// TwinCAT 3 PLC project rixs_optics
// ProgramVersion: 3.1.4022.7
// libraries:
//   lcls2-cc-lib, * (SLAC)
//   PMPS, * (SLAC - LCLS)
//   Tc2_MC2, * (Beckhoff Automation GmbH)
//   Tc2_SerialCom, * (Beckhoff Automation GmbH)
//   Tc2_Standard, * (Beckhoff Automation GmbH)
//   Tc2_System, * (Beckhoff Automation GmbH)
//   Tc2_Utilities, * (Beckhoff Automation GmbH)
//   Tc3_Module, * (Beckhoff Automation GmbH)
//   LCLS General,newest,SLAC
//   lcls-twincat-motion,newest,SLAC
//   lcls-twincat-optics,newest,SLAC
// project tree:
//   DUTs/ ENUM_XS_YAG_States.TcDUT (not stored)
//   Function Blocks/ FB_XS_YAG_States.TcPOU (not stored)
//   GVLs/ GVL_COM_Buffers.TcGVL (not stored), GVL_M1K1.TcGVL (not stored), GVL_M1K1_BENDER_Constants.TcGVL (not stored), GVL_M1K1_BENDER_RTD.TcGVL (not stored), GVL_M1K1_Constants.TcGVL (not stored), GVL_M1K2.TcGVL (not stored), GVL_M1K2_Constants.TcGVL (not stored), GVL_PMPS.TcGVL (not stored), GVL_SerialIO.TcGVL (not stored), Main.TcGVL
//   / PiezoDriver.TcTTO (not stored), PlcTask.TcTTO (not stored), SerialIO.TcTTO (not stored)
//   POUs/ PRG_1_PlcTask.TcPOU (not stored), PRG_2_PMPS_POST.TcPOU (not stored), PRG_MR1K1_BEND.TcPOU (not stored), PRG_MR1K1_BEND_BENDER.TcPOU (not stored), PRG_MR1K2_SWITCH.TcPOU (not stored), PRG_SL1K2_EXIT.TcPOU (not stored), PRG_SP1K1_MONO.TcPOU (not stored), PRG_SPO_PMPS.TcPOU, PRG_ST1K1_ZOS.TcPOU (not stored)
//   POUs/Serial Comm/ PiezoSerial.TcPOU (not stored), P_Serial_Com.TcPOU (not stored)
// real-time tasks:
//   TASK PlcTask: cycle T#10ms, priority 20, ADS port 350
//   TASK PiezoDriver: cycle T#1ms, priority 3, ADS port 351
//   TASK SerialIO: cycle T#2ms, priority 1, ADS port 352
// motion (NC):
// I/O:
//   DEVICE Device 1 (EtherCAT)
// variable links:
//   rixs_optics Instance <-> Device 1 (EtherCAT)/Term 1 (EK1200)/E5 (EK1122)/Box 84 (EP2338-0002)
//     PlcTask Outputs/PRG_SP1K1_MONO.bLEDPower01 <-> Channel 10/Output
//     PlcTask Outputs/PRG_SP1K1_MONO.bLEDPower02 <-> Channel 12/Output
//     PlcTask Outputs/PRG_SP1K1_MONO.bLEDPower03 <-> Channel 14/Output
//   rixs_optics Instance <-> Device 1 (EtherCAT)/Term 1 (EK1200)/E5 (EK1122)/SL1K2-EXIT (EK1100)/EL2004_SL1K2
//     PlcTask Outputs/PRG_SL1K2_EXIT.bFanOn <-> Channel 1/Output
//     PlcTask Outputs/PRG_SL1K2_EXIT.bLEDPower <-> Channel 2/Output
//     PlcTask Outputs/PRG_SL1K2_EXIT.fbGige.bGigePower <-> Channel 3/Output
//   rixs_optics Instance <-> Device 1 (EtherCAT)/Term 1 (EK1200)/E5 (EK1122)/SL1K2-EXIT (EK1100)/EL3201_SL1K2_1
//     PlcTask Inputs/PRG_SL1K2_EXIT.RTD_Crystal_TOP.bOverrange <-> RTD/Status/Overrange
//     PlcTask Inputs/PRG_SL1K2_EXIT.RTD_Crystal_TOP.bUnderrange <-> RTD/Status/Underrange
//     PlcTask Inputs/PRG_SL1K2_EXIT.RTD_Crystal_TOP.iRaw <-> RTD/Value
//   rixs_optics Instance <-> Device 1 (EtherCAT)/Term 1 (EK1200)/E5 (EK1122)/SL1K2-EXIT (EK1100)/EL3201_SL1K2_2
//     PlcTask Inputs/PRG_SL1K2_EXIT.RTD_Crystal_BOTTOM.bOverrange <-> RTD/Status/Overrange
//     PlcTask Inputs/PRG_SL1K2_EXIT.RTD_Crystal_BOTTOM.bUnderrange <-> RTD/Status/Underrange
//     PlcTask Inputs/PRG_SL1K2_EXIT.RTD_Crystal_BOTTOM.iRaw <-> RTD/Value
//   rixs_optics Instance <-> Device 1 (EtherCAT)/Term 1 (EK1200)/E5 (EK1122)/SL1K2-EXIT (EK1100)/EL3201_SL1K2_3
//     PlcTask Inputs/PRG_SL1K2_EXIT.RTD_YAG.bOverrange <-> RTD/Status/Overrange
//     PlcTask Inputs/PRG_SL1K2_EXIT.RTD_YAG.bUnderrange <-> RTD/Status/Underrange
//     PlcTask Inputs/PRG_SL1K2_EXIT.RTD_YAG.iRaw <-> RTD/Value
//   rixs_optics Instance <-> Device 1 (EtherCAT)/Term 1 (EK1200)/E5 (EK1122)/SL1K2-EXIT (EK1100)/EL3201_SL1K2_4
//     PlcTask Inputs/PRG_SL1K2_EXIT.RTD_HeatSync.bOverrange <-> RTD/Status/Overrange
//     PlcTask Inputs/PRG_SL1K2_EXIT.RTD_HeatSync.bUnderrange <-> RTD/Status/Underrange
//     PlcTask Inputs/PRG_SL1K2_EXIT.RTD_HeatSync.iRaw <-> RTD/Value
//   rixs_optics Instance <-> Device 1 (EtherCAT)/Term 1 (EK1200)/E5 (EK1122)/SL1K2-EXIT (EK1100)/EL4004_SL1K2
//     PlcTask Outputs/PRG_SL1K2_EXIT.fbGige.iIlluminatorINT <-> AO Outputs Channel 1/Analog output
//   rixs_optics Instance <-> Device 1 (EtherCAT)/Term 1 (EK1200)/E5 (EK1122)/SL1K2-EXIT (EK1100)/EL5042_SL1K2_PITCH_VERT
//     PlcTask Inputs/Main.M19.nRawEncoderUINT <-> FB Inputs Channel 1/Position
//     PlcTask Inputs/Main.M20.nRawEncoderUINT <-> FB Inputs Channel 2/Position
//   rixs_optics Instance <-> Device 1 (EtherCAT)/Term 1 (EK1200)/E5 (EK1122)/SL1K2-EXIT (EK1100)/EL5042_SL1K2_ROLL_GAP
//     PlcTask Inputs/Main.M21.nRawEncoderUINT <-> FB Inputs Channel 1/Position
//     PlcTask Inputs/Main.M22.nRawEncoderUINT <-> FB Inputs Channel 2/Position
//   rixs_optics Instance <-> Device 1 (EtherCAT)/Term 1 (EK1200)/E5 (EK1122)/SL1K2-EXIT (EK1100)/EL5042_SL1K2_YAG
//     PlcTask Inputs/Main.M23.nRawEncoderUINT <-> FB Inputs Channel 1/Position
//   rixs_optics Instance <-> Device 1 (EtherCAT)/Term 1 (EK1200)/E5 (EK1122)/SL1K2-EXIT (EK1100)/EL7047_SL1K2_GAP
//     PlcTask Inputs/Main.M22.bLimitBackwardEnable <-> STM Status/Status/Digital input 1
//     PlcTask Inputs/Main.M22.bLimitForwardEnable <-> STM Status/Status/Digital input 2
//   rixs_optics Instance <-> Device 1 (EtherCAT)/Term 1 (EK1200)/E5 (EK1122)/SL1K2-EXIT (EK1100)/EL7047_SL1K2_PITCH
//     PlcTask Inputs/Main.M19.bLimitBackwardEnable <-> STM Status/Status/Digital input 1
//     PlcTask Inputs/Main.M19.bLimitForwardEnable <-> STM Status/Status/Digital input 2
//   rixs_optics Instance <-> Device 1 (EtherCAT)/Term 1 (EK1200)/E5 (EK1122)/SL1K2-EXIT (EK1100)/EL7047_SL1K2_ROLL
//     PlcTask Inputs/Main.M21.bLimitBackwardEnable <-> STM Status/Status/Digital input 1
//     PlcTask Inputs/Main.M21.bLimitForwardEnable <-> STM Status/Status/Digital input 2
//   rixs_optics Instance <-> Device 1 (EtherCAT)/Term 1 (EK1200)/E5 (EK1122)/SL1K2-EXIT (EK1100)/EL7047_SL1K2_VERT
//     PlcTask Inputs/Main.M20.bLimitBackwardEnable <-> STM Status/Status/Digital input 2
//     PlcTask Inputs/Main.M20.bLimitForwardEnable <-> STM Status/Status/Digital input 1
//   rixs_optics Instance <-> Device 1 (EtherCAT)/Term 1 (EK1200)/E5 (EK1122)/SL1K2-EXIT (EK1100)/EL7047_SL1K2_YAG
//     PlcTask Inputs/Main.M23.bLimitBackwardEnable <-> STM Status/Status/Digital input 2
//     PlcTask Inputs/Main.M23.bLimitForwardEnable <-> STM Status/Status/Digital input 1
//   rixs_optics Instance <-> Device 1 (EtherCAT)/Term 1 (EK1200)/E5 (EK1122)/X1 SP1K1-MONO(EK1100)/SP1K1-EL1004-E17
//     PlcTask Inputs/PRG_SP1K1_MONO.bSTOEnable1 <-> Channel 1/Input
//     PlcTask Inputs/PRG_SP1K1_MONO.bSTOEnable2 <-> Channel 2/Input
//   rixs_optics Instance <-> Device 1 (EtherCAT)/Term 1 (EK1200)/E5 (EK1122)/X1 SP1K1-MONO(EK1100)/SP1K1-EL3054-E12
//     PlcTask Inputs/PRG_SP1K1_MONO.flow_1 <-> AI Standard Channel 1/Value
//     PlcTask Inputs/PRG_SP1K1_MONO.flow_2 <-> AI Standard Channel 2/Value
//     PlcTask Inputs/PRG_SP1K1_MONO.pres_1 <-> AI Standard Channel 3/Value
//   rixs_optics Instance <-> Device 1 (EtherCAT)/Term 1 (EK1200)/E5 (EK1122)/X1 SP1K1-MONO(EK1100)/SP1K1-EL3202-E13
//     PlcTask Inputs/PRG_SP1K1_MONO.RTD1.bError <-> RTD Inputs Channel 1/Status/Error
//     PlcTask Inputs/PRG_SP1K1_MONO.RTD2.bError <-> RTD Inputs Channel 2/Status/Error
//     PlcTask Inputs/PRG_SP1K1_MONO.RTD1.bOverrange <-> RTD Inputs Channel 1/Status/Overrange
//     PlcTask Inputs/PRG_SP1K1_MONO.RTD2.bOverrange <-> RTD Inputs Channel 2/Status/Overrange
//     PlcTask Inputs/PRG_SP1K1_MONO.RTD1.bUnderrange <-> RTD Inputs Channel 1/Status/Underrange
//     PlcTask Inputs/PRG_SP1K1_MONO.RTD2.bUnderrange <-> RTD Inputs Channel 2/Status/Underrange
//     PlcTask Inputs/PRG_SP1K1_MONO.RTD1.iRaw <-> RTD Inputs Channel 1/Value
//     PlcTask Inputs/PRG_SP1K1_MONO.RTD2.iRaw <-> RTD Inputs Channel 2/Value
//   rixs_optics Instance <-> Device 1 (EtherCAT)/Term 1 (EK1200)/E5 (EK1122)/X1 SP1K1-MONO(EK1100)/SP1K1-EL3202-E14
//     PlcTask Inputs/PRG_SP1K1_MONO.RTD3.bError <-> RTD Inputs Channel 1/Status/Error
//     PlcTask Inputs/PRG_SP1K1_MONO.RTD4.bError <-> RTD Inputs Channel 2/Status/Error
//     PlcTask Inputs/PRG_SP1K1_MONO.RTD3.bOverrange <-> RTD Inputs Channel 1/Status/Overrange
//     PlcTask Inputs/PRG_SP1K1_MONO.RTD4.bOverrange <-> RTD Inputs Channel 2/Status/Overrange
//     PlcTask Inputs/PRG_SP1K1_MONO.RTD3.bUnderrange <-> RTD Inputs Channel 1/Status/Underrange
//     PlcTask Inputs/PRG_SP1K1_MONO.RTD4.bUnderrange <-> RTD Inputs Channel 2/Status/Underrange
//     PlcTask Inputs/PRG_SP1K1_MONO.RTD3.iRaw <-> RTD Inputs Channel 1/Value
//     PlcTask Inputs/PRG_SP1K1_MONO.RTD4.iRaw <-> RTD Inputs Channel 2/Value
//   rixs_optics Instance <-> Device 1 (EtherCAT)/Term 1 (EK1200)/E5 (EK1122)/X1 SP1K1-MONO(EK1100)/SP1K1-EL3204-E15
//     PlcTask Inputs/PRG_SP1K1_MONO.RTD5.bError <-> RTD Inputs Channel 1/Status/Error
//     PlcTask Inputs/PRG_SP1K1_MONO.RTD6.bError <-> RTD Inputs Channel 2/Status/Error
//     PlcTask Inputs/PRG_SP1K1_MONO.RTD5.bOverrange <-> RTD Inputs Channel 1/Status/Overrange
//     PlcTask Inputs/PRG_SP1K1_MONO.RTD6.bOverrange <-> RTD Inputs Channel 2/Status/Overrange
//     PlcTask Inputs/PRG_SP1K1_MONO.RTD5.bUnderrange <-> RTD Inputs Channel 1/Status/Underrange
//     PlcTask Inputs/PRG_SP1K1_MONO.RTD6.bUnderrange <-> RTD Inputs Channel 2/Status/Underrange
//     PlcTask Inputs/PRG_SP1K1_MONO.RTD5.iRaw <-> RTD Inputs Channel 1/Value
//     PlcTask Inputs/PRG_SP1K1_MONO.RTD6.iRaw <-> RTD Inputs Channel 2/Value
//   rixs_optics Instance <-> Device 1 (EtherCAT)/Term 1 (EK1200)/E5 (EK1122)/X1 SP1K1-MONO(EK1100)/SP1K1-EL3204-E16
//     PlcTask Inputs/PRG_SP1K1_MONO.RTD7.bError <-> RTD Inputs Channel 1/Status/Error
//     PlcTask Inputs/PRG_SP1K1_MONO.RTD8.bError <-> RTD Inputs Channel 2/Status/Error
//     PlcTask Inputs/PRG_SP1K1_MONO.RTD7.bOverrange <-> RTD Inputs Channel 1/Status/Overrange
//     PlcTask Inputs/PRG_SP1K1_MONO.RTD8.bOverrange <-> RTD Inputs Channel 2/Status/Overrange
//     PlcTask Inputs/PRG_SP1K1_MONO.RTD7.bUnderrange <-> RTD Inputs Channel 1/Status/Underrange
//     PlcTask Inputs/PRG_SP1K1_MONO.RTD8.bUnderrange <-> RTD Inputs Channel 2/Status/Underrange
//     PlcTask Inputs/PRG_SP1K1_MONO.RTD7.iRaw <-> RTD Inputs Channel 1/Value
//     PlcTask Inputs/PRG_SP1K1_MONO.RTD8.iRaw <-> RTD Inputs Channel 2/Value
//   rixs_optics Instance <-> Device 1 (EtherCAT)/Term 1 (EK1200)/E5 (EK1122)/X1 SP1K1-MONO(EK1100)/g_h_m
//     PlcTask Inputs/Main.M9.bLimitBackwardEnable <-> STM Status/Status/Digital input 2
//     PlcTask Inputs/Main.M9.bLimitForwardEnable <-> STM Status/Status/Digital input 1
//   rixs_optics Instance <-> Device 1 (EtherCAT)/Term 1 (EK1200)/E5 (EK1122)/X1 SP1K1-MONO(EK1100)/g_pi_m
//     PlcTask Inputs/Main.M7.bLimitBackwardEnable <-> STM Status/Status/Digital input 2
//     PlcTask Inputs/Main.M7.bLimitForwardEnable <-> STM Status/Status/Digital input 1
//   rixs_optics Instance <-> Device 1 (EtherCAT)/Term 1 (EK1200)/E5 (EK1122)/X1 SP1K1-MONO(EK1100)/g_pi_up_dwn_e
//     PlcTask Inputs/PRG_SP1K1_MONO.gpi_upe/Count <-> FB Inputs Channel 1/Position
//   rixs_optics Instance <-> Device 1 (EtherCAT)/Term 1 (EK1200)/E5 (EK1122)/X1 SP1K1-MONO(EK1100)/m_h_m
//     PlcTask Inputs/Main.M8.bLimitBackwardEnable <-> STM Status/Status/Digital input 2
//     PlcTask Inputs/Main.M8.bLimitForwardEnable <-> STM Status/Status/Digital input 1
//   rixs_optics Instance <-> Device 1 (EtherCAT)/Term 1 (EK1200)/E5 (EK1122)/X1 SP1K1-MONO(EK1100)/m_pi_m
//     PlcTask Inputs/Main.M6.bLimitBackwardEnable <-> STM Status/Status/Digital input 2
//     PlcTask Inputs/Main.M6.bLimitForwardEnable <-> STM Status/Status/Digital input 1
//   rixs_optics Instance <-> Device 1 (EtherCAT)/Term 1 (EK1200)/E5 (EK1122)/X1 SP1K1-MONO(EK1100)/m_pi_up_dwn_e
//     PlcTask Inputs/PRG_SP1K1_MONO.mpi_upe/Count <-> FB Inputs Channel 1/Position
//   rixs_optics Instance <-> Device 1 (EtherCAT)/Term 1 (EK1200)/E5 (EK1122)/X1 SP1K1-MONO(EK1100)/s_io_m
//     PlcTask Inputs/Main.M10.bLimitBackwardEnable <-> STM Status/Status/Digital input 2
//     PlcTask Inputs/Main.M10.bLimitForwardEnable <-> STM Status/Status/Digital input 1
//     PlcTask Inputs/Main.sio_current <-> STM Synchron info data/Info data 1
//     PlcTask Inputs/Main.sio_load <-> STM Synchron info data/Info data 2
//   rixs_optics Instance <-> Device 1 (EtherCAT)/Term 1 (EK1200)/PMPS_FFO
//     PlcTask Outputs/GVL_PMPS.fbFastFaultOutput1.q_xFastFaultOut <-> Channel 1/Output
//     PlcTask Outputs/GVL_PMPS.fbFastFaultOutput2.q_xFastFaultOut <-> Channel 2/Output
//   rixs_optics Instance <-> Device 1 (EtherCAT)/Term 1 (EK1200)/PMPS_PRE
//     PlcTask Inputs/PRG_2_PMPS_POST.fbArbiterIO.i_stCurrentBP <-> IO Inputs/CurrentBP
//     PlcTask Inputs/PRG_2_PMPS_POST.fbArbiterIO.xTxPDO_state <-> SYNC Inputs/TxPDO state
//     PlcTask Inputs/PRG_2_PMPS_POST.fbArbiterIO.xTxPDO_toggle <-> SYNC Inputs/TxPDO toggle
//     PlcTask Outputs/PRG_2_PMPS_POST.fbArbiterIO.q_stRequestedBP <-> IO Outputs/RequestedBP
//     PlcTask Outputs/PRG_MR1K1_BEND.nMR1K1_Y_ENC_PMPS <-> IO Outputs/MR1K1_Y_ENC
//   rixs_optics Instance <-> Device 1 (EtherCAT)/Term 1 (EK1200)/Term 5 (EK1122)/EK1100_M1K2/EL1004_M1K2_STO
//     PlcTask Inputs/PRG_MR1K2_SWITCH.M1K2.fbRunHOMS.bSTOEnable1 <-> Channel 1/Input
//     PlcTask Inputs/PRG_MR1K2_SWITCH.M1K2.fbRunHOMS.bSTOEnable2 <-> Channel 2/Input
//   rixs_optics Instance <-> Device 1 (EtherCAT)/Term 1 (EK1200)/Term 5 (EK1122)/EK1100_M1K2/EL5042_M1K2_Pitch
//     PlcTask Inputs/GVL_M1K1.M1K1_Pitch.diEncCnt <-> FB Inputs Channel 1/Position
//     PlcTask Inputs/GVL_M1K2.M1K2_Pitch.diEncCnt <-> FB Inputs Channel 1/Position
//   rixs_optics Instance <-> Device 1 (EtherCAT)/Term 1 (EK1200)/Term 5 (EK1122)/EK1100_M1K2/EL5042_M1K2_Xupdwn
//     PlcTask Inputs/PRG_MR1K2_SWITCH.M1K2.fbRunHOMS.stXdwnEnc/Count <-> FB Inputs Channel 2/Position
//     PlcTask Inputs/PRG_MR1K2_SWITCH.M1K2.fbRunHOMS.stXupEnc/Count <-> FB Inputs Channel 1/Position
//   rixs_optics Instance <-> Device 1 (EtherCAT)/Term 1 (EK1200)/Term 5 (EK1122)/EK1100_M1K2/EL5042_M1K2_Yleftright
//     PlcTask Inputs/PRG_MR1K2_SWITCH.M1K2.fbRunHOMS.stYdwnEnc/Count <-> FB Inputs Channel 2/Position
//     PlcTask Inputs/PRG_MR1K2_SWITCH.M1K2.fbRunHOMS.stYupEnc/Count <-> FB Inputs Channel 1/Position
//   rixs_optics Instance <-> Device 1 (EtherCAT)/Term 1 (EK1200)/Term 5 (EK1122)/EK1100_M1K2/EL6001_M1K2_PitchFine
//     SerialIO Inputs/GVL_SerialIO.Serial_stComIn_M1K2/D[{0..21}] <-> COM Inputs/Data In {0..21}  (22 links)
//     SerialIO Inputs/GVL_SerialIO.Serial_stComIn_M1K2/Status <-> COM Inputs/Status
//     SerialIO Outputs/GVL_SerialIO.Serial_stComOut_M1K2/Ctrl <-> COM Outputs/Ctrl
//     SerialIO Outputs/GVL_SerialIO.Serial_stComOut_M1K2/D[{0..21}] <-> COM Outputs/Data Out {0..21}  (22 links)
//   rixs_optics Instance <-> Device 1 (EtherCAT)/Term 1 (EK1200)/Term 5 (EK1122)/EK1100_M1K2/EL7047_M1K2_PitchCoarse
//     PlcTask Inputs/Main.M5.bLimitBackwardEnable <-> STM Status/Status/Digital input 2
//     PlcTask Inputs/Main.M5.bLimitForwardEnable <-> STM Status/Status/Digital input 1
//   rixs_optics Instance <-> Device 1 (EtherCAT)/Term 1 (EK1200)/Term 5 (EK1122)/EK1100_M1K2/EL7047_M1K2_Xdwn
//     PlcTask Inputs/Main.M4.bLimitBackwardEnable <-> STM Status/Status/Digital input 2
//     PlcTask Inputs/Main.M4.bLimitForwardEnable <-> STM Status/Status/Digital input 1
//   rixs_optics Instance <-> Device 1 (EtherCAT)/Term 1 (EK1200)/Term 5 (EK1122)/EK1100_M1K2/EL7047_M1K2_Xup
//     PlcTask Inputs/Main.M3.bLimitBackwardEnable <-> STM Status/Status/Digital input 2
//     PlcTask Inputs/Main.M3.bLimitForwardEnable <-> STM Status/Status/Digital input 1
//   rixs_optics Instance <-> Device 1 (EtherCAT)/Term 1 (EK1200)/Term 5 (EK1122)/EK1100_M1K2/EL7047_M1K2_Yleft
//     PlcTask Inputs/Main.M1.bLimitBackwardEnable <-> STM Status/Status/Digital input 2
//     PlcTask Inputs/Main.M1.bLimitForwardEnable <-> STM Status/Status/Digital input 1
//   rixs_optics Instance <-> Device 1 (EtherCAT)/Term 1 (EK1200)/Term 5 (EK1122)/EK1100_M1K2/EL7047_M1K2_Yright
//     PlcTask Inputs/Main.M2.bLimitBackwardEnable <-> STM Status/Status/Digital input 2
//     PlcTask Inputs/Main.M2.bLimitForwardEnable <-> STM Status/Status/Digital input 1
//   rixs_optics Instance <-> Device 1 (EtherCAT)/Term 1 (EK1200)/Term 5 (EK1122)/EK1100_MR1K1/EL1004_M1K1_STO
//     PlcTask Inputs/PRG_MR1K1_BEND.M1K1.fbRunHOMS.bSTOEnable1 <-> Channel 1/Input
//     PlcTask Inputs/PRG_MR1K1_BEND.M1K1.fbRunHOMS.bSTOEnable2 <-> Channel 2/Input
//   rixs_optics Instance <-> Device 1 (EtherCAT)/Term 1 (EK1200)/Term 5 (EK1122)/EK1100_MR1K1/EL5042_M1K1_Xupdwn
//     PlcTask Inputs/PRG_MR1K1_BEND.M1K1.fbRunHOMS.stXdwnEnc/Count <-> FB Inputs Channel 2/Position
//     PlcTask Inputs/PRG_MR1K1_BEND.M1K1.fbRunHOMS.stXupEnc/Count <-> FB Inputs Channel 1/Position
//   rixs_optics Instance <-> Device 1 (EtherCAT)/Term 1 (EK1200)/Term 5 (EK1122)/EK1100_MR1K1/EL5042_M1K1_Yupdwn
//     PlcTask Inputs/PRG_MR1K1_BEND.M1K1.fbRunHOMS.stYdwnEnc/Count <-> FB Inputs Channel 2/Position
//     PlcTask Inputs/PRG_MR1K1_BEND.M1K1.fbRunHOMS.stYupEnc/Count <-> FB Inputs Channel 1/Position
//     PlcTask Inputs/PRG_MR1K1_BEND.bMR1K1_Y_ENC_Ready <-> FB Inputs Channel 1/Status/Ready
//     PlcTask Inputs/PRG_MR1K1_BEND.bMR1K1_Y_ENC_TxPDO <-> FB Inputs Channel 1/Status/TxPDO State
//   rixs_optics Instance <-> Device 1 (EtherCAT)/Term 1 (EK1200)/Term 5 (EK1122)/EK1100_MR1K1/EL7047_M1K1_PitchCoarse
//     PlcTask Inputs/Main.M16.bLimitBackwardEnable <-> STM Status/Status/Digital input 2
//     PlcTask Inputs/Main.M16.bLimitForwardEnable <-> STM Status/Status/Digital input 1
//   rixs_optics Instance <-> Device 1 (EtherCAT)/Term 1 (EK1200)/Term 5 (EK1122)/EK1100_MR1K1/EL7047_M1K1_Xdwn
//     PlcTask Inputs/Main.M15.bLimitBackwardEnable <-> STM Status/Status/Digital input 2
//     PlcTask Inputs/Main.M15.bLimitForwardEnable <-> STM Status/Status/Digital input 1
//   rixs_optics Instance <-> Device 1 (EtherCAT)/Term 1 (EK1200)/Term 5 (EK1122)/EK1100_MR1K1/EL7047_M1K1_Xup
//     PlcTask Inputs/Main.M14.bLimitBackwardEnable <-> STM Status/Status/Digital input 2
//     PlcTask Inputs/Main.M14.bLimitForwardEnable <-> STM Status/Status/Digital input 1
//   rixs_optics Instance <-> Device 1 (EtherCAT)/Term 1 (EK1200)/Term 5 (EK1122)/EK1100_MR1K1/EL7047_M1K1_Ydwn
//     PlcTask Inputs/Main.M12.bLimitBackwardEnable <-> STM Status/Status/Digital input 2
//     PlcTask Inputs/Main.M13.bLimitBackwardEnable <-> STM Status/Status/Digital input 2
//     PlcTask Inputs/Main.M13.bLimitForwardEnable <-> STM Status/Status/Digital input 1
//   rixs_optics Instance <-> Device 1 (EtherCAT)/Term 1 (EK1200)/Term 5 (EK1122)/EK1100_MR1K1/EL7047_M1K1_Yup
//     PlcTask Inputs/Main.M12.bLimitForwardEnable <-> STM Status/Status/Digital input 1
//   rixs_optics Instance <-> Device 1 (EtherCAT)/Term 1 (EK1200)/Term 5 (EK1122)/EK1100_MR1K1_BEND/EL1004_M1K1_BENDER_STO
//     PlcTask Inputs/PRG_MR1K1_BEND_BENDER.M1K1BENDbSTOEnable1 <-> Channel 1/Input
//     PlcTask Inputs/PRG_MR1K1_BEND_BENDER.M1K1BENDbSTOEnable2 <-> Channel 2/Input
//   rixs_optics Instance <-> Device 1 (EtherCAT)/Term 1 (EK1200)/Term 5 (EK1122)/EK1100_MR1K1_BEND/EL2024-0010_M1K1_BEND_LED1
//     PlcTask Outputs/PRG_MR1K1_BEND.bLEDPower01 <-> Channel 1/Output
//     PlcTask Outputs/PRG_MR1K1_BEND.bLEDPower02 <-> Channel 2/Output
//     PlcTask Outputs/PRG_MR1K1_BEND.bLEDPower03 <-> Channel 3/Output
//     PlcTask Outputs/PRG_MR1K1_BEND.bLEDPower04 <-> Channel 4/Output
//   rixs_optics Instance <-> Device 1 (EtherCAT)/Term 1 (EK1200)/Term 5 (EK1122)/EK1100_MR1K1_BEND/EL3202-0010_M1K1DS2_M1K1DS3
//     PlcTask Inputs/GVL_M1K1_BENDER_RTD.nM1K1DS_RTD_2 <-> RTD Inputs Channel 1/Value
//     PlcTask Inputs/GVL_M1K1_BENDER_RTD.nM1K1DS_RTD_3 <-> RTD Inputs Channel 2/Value
//   rixs_optics Instance <-> Device 1 (EtherCAT)/Term 1 (EK1200)/Term 5 (EK1122)/EK1100_MR1K1_BEND/EL3202-0010_M1K1US1_M1K1US2
//     PlcTask Inputs/GVL_M1K1_BENDER_RTD.nM1K1US_RTD_1 <-> RTD Inputs Channel 1/Value
//     PlcTask Inputs/GVL_M1K1_BENDER_RTD.nM1K1US_RTD_2 <-> RTD Inputs Channel 2/Value
//   rixs_optics Instance <-> Device 1 (EtherCAT)/Term 1 (EK1200)/Term 5 (EK1122)/EK1100_MR1K1_BEND/EL3202-0010_M1K1US3_M1K1DS1
//     PlcTask Inputs/GVL_M1K1_BENDER_RTD.nM1K1DS_RTD_1 <-> RTD Inputs Channel 2/Value
//     PlcTask Inputs/GVL_M1K1_BENDER_RTD.nM1K1US_RTD_3 <-> RTD Inputs Channel 1/Value
//   rixs_optics Instance <-> Device 1 (EtherCAT)/Term 1 (EK1200)/Term 5 (EK1122)/EK1100_MR1K1_BEND/EL5042_M1K1_BEND_USDS
//     PlcTask Inputs/Main.M17.nRawEncoderULINT <-> FB Inputs Channel 1/Position
//     PlcTask Inputs/Main.M18.nRawEncoderULINT <-> FB Inputs Channel 2/Position
//   rixs_optics Instance <-> Device 1 (EtherCAT)/Term 1 (EK1200)/Term 5 (EK1122)/EK1100_MR1K1_BEND/EL7041_M1K1_BEND_DS
//     PlcTask Inputs/Main.M18.bLimitBackwardEnable <-> STM Status/Status/Digital input 2
//     PlcTask Inputs/Main.M18.bLimitForwardEnable <-> STM Status/Status/Digital input 1
//   rixs_optics Instance <-> Device 1 (EtherCAT)/Term 1 (EK1200)/Term 5 (EK1122)/EK1100_MR1K1_BEND/EL7041_M1K1_BEND_US
//     PlcTask Inputs/Main.M17.bLimitBackwardEnable <-> STM Status/Status/Digital input 2
//     PlcTask Inputs/Main.M17.bLimitForwardEnable <-> STM Status/Status/Digital input 1
//   rixs_optics Instance <-> Device 1 (EtherCAT)/Term 1 (EK1200)/Term 5 (EK1122)/EK1100_ST1K2_ZOS/ST1K1-EL2008
//     PlcTask Outputs/Main.M24.bBrakeRelease <-> Channel 1/Output
//   rixs_optics Instance <-> Device 1 (EtherCAT)/Term 1 (EK1200)/Term 5 (EK1122)/EK1100_ST1K2_ZOS/ST1K1-EL7041
//     PlcTask Inputs/Main.M24.bLimitBackwardEnable <-> STM Status/Status/Digital input 2
//     PlcTask Inputs/Main.M24.bLimitForwardEnable <-> STM Status/Status/Digital input 1
//   rixs_optics Instance <-> NC-Task 1 SAF/Axes/Axis 24 ST1K1-ZOS-MMS
//     PlcTask Inputs/Main.M24.Axis.NcToPlc <-> Outputs/ToPlc
//     PlcTask Outputs/Main.M24.Axis.PlcToNc <-> Inputs/FromPlc
//   rixs_optics Instance <-> NC-Task 1 SAF/Axes/M1K1-BEND-DS
//     PlcTask Inputs/Main.M18.Axis.NcToPlc <-> Outputs/ToPlc
//     PlcTask Outputs/Main.M18.Axis.PlcToNc <-> Inputs/FromPlc
//   rixs_optics Instance <-> NC-Task 1 SAF/Axes/M1K1-BEND-US
//     PlcTask Inputs/Main.M17.Axis.NcToPlc <-> Outputs/ToPlc
//     PlcTask Outputs/Main.M17.Axis.PlcToNc <-> Inputs/FromPlc
//   rixs_optics Instance <-> NC-Task 1 SAF/Axes/M1K1-Pitch
//     PlcTask Inputs/Main.M16.Axis.NcToPlc <-> Outputs/ToPlc
//     PlcTask Outputs/Main.M16.Axis.PlcToNc <-> Inputs/FromPlc
//   rixs_optics Instance <-> NC-Task 1 SAF/Axes/M1K1-Xdwn
//     PlcTask Inputs/Main.M15.Axis.NcToPlc <-> Outputs/ToPlc
//     PlcTask Outputs/Main.M15.Axis.PlcToNc <-> Inputs/FromPlc
//   rixs_optics Instance <-> NC-Task 1 SAF/Axes/M1K1-Xup
//     PlcTask Inputs/Main.M14.Axis.NcToPlc <-> Outputs/ToPlc
//     PlcTask Outputs/Main.M14.Axis.PlcToNc <-> Inputs/FromPlc
//   rixs_optics Instance <-> NC-Task 1 SAF/Axes/M1K1-Ydwn
//     PlcTask Inputs/Main.M13.Axis.NcToPlc <-> Outputs/ToPlc
//     PlcTask Outputs/Main.M13.Axis.PlcToNc <-> Inputs/FromPlc
//   rixs_optics Instance <-> NC-Task 1 SAF/Axes/M1K1-Yup
//     PlcTask Inputs/Main.M12.Axis.NcToPlc <-> Outputs/ToPlc
//     PlcTask Outputs/Main.M12.Axis.PlcToNc <-> Inputs/FromPlc
//   rixs_optics Instance <-> NC-Task 1 SAF/Axes/M1K2-Pitch
//     PlcTask Inputs/Main.M5.Axis.NcToPlc <-> Outputs/ToPlc
//     PlcTask Outputs/Main.M5.Axis.PlcToNc <-> Inputs/FromPlc
//   rixs_optics Instance <-> NC-Task 1 SAF/Axes/M1K2-Xdwn
//     PlcTask Inputs/Main.M4.Axis.NcToPlc <-> Outputs/ToPlc
//     PlcTask Outputs/Main.M4.Axis.PlcToNc <-> Inputs/FromPlc
//   rixs_optics Instance <-> NC-Task 1 SAF/Axes/M1K2-Xup
//     PlcTask Inputs/Main.M3.Axis.NcToPlc <-> Outputs/ToPlc
//     PlcTask Outputs/Main.M3.Axis.PlcToNc <-> Inputs/FromPlc
//   rixs_optics Instance <-> NC-Task 1 SAF/Axes/M1K2-Yleft
//     PlcTask Inputs/Main.M1.Axis.NcToPlc <-> Outputs/ToPlc
//     PlcTask Outputs/Main.M1.Axis.PlcToNc <-> Inputs/FromPlc
//   rixs_optics Instance <-> NC-Task 1 SAF/Axes/M1K2-Yright
//     PlcTask Inputs/Main.M2.Axis.NcToPlc <-> Outputs/ToPlc
//     PlcTask Outputs/Main.M2.Axis.PlcToNc <-> Inputs/FromPlc
//   rixs_optics Instance <-> NC-Task 1 SAF/Axes/SL1K2-CrystalGap-M22
//     PlcTask Inputs/Main.M22.Axis.NcToPlc <-> Outputs/ToPlc
//     PlcTask Outputs/Main.M22.Axis.PlcToNc <-> Inputs/FromPlc
//   rixs_optics Instance <-> NC-Task 1 SAF/Axes/SL1K2-Pitch-M19
//     PlcTask Inputs/Main.M19.Axis.NcToPlc <-> Outputs/ToPlc
//     PlcTask Outputs/Main.M19.Axis.PlcToNc <-> Inputs/FromPlc
//   rixs_optics Instance <-> NC-Task 1 SAF/Axes/SL1K2-Roll-M21
//     PlcTask Inputs/Main.M21.Axis.NcToPlc <-> Outputs/ToPlc
//     PlcTask Outputs/Main.M21.Axis.PlcToNc <-> Inputs/FromPlc
//   rixs_optics Instance <-> NC-Task 1 SAF/Axes/SL1K2-Vert-M20
//     PlcTask Inputs/Main.M20.Axis.NcToPlc <-> Outputs/ToPlc
//     PlcTask Outputs/Main.M20.Axis.PlcToNc <-> Inputs/FromPlc
//   rixs_optics Instance <-> NC-Task 1 SAF/Axes/SL1K2-YAG-M23
//     PlcTask Inputs/Main.M23.Axis.NcToPlc <-> Outputs/ToPlc
//     PlcTask Outputs/Main.M23.Axis.PlcToNc <-> Inputs/FromPlc
//   rixs_optics Instance <-> NC-Task 1 SAF/Axes/g_h
//     PlcTask Inputs/Main.M9.Axis.NcToPlc <-> Outputs/ToPlc
//     PlcTask Outputs/Main.M9.Axis.PlcToNc <-> Inputs/FromPlc
//   rixs_optics Instance <-> NC-Task 1 SAF/Axes/g_pi
//     PlcTask Inputs/Main.M7.Axis.NcToPlc <-> Outputs/ToPlc
//     PlcTask Outputs/Main.M7.Axis.PlcToNc <-> Inputs/FromPlc
//   rixs_optics Instance <-> NC-Task 1 SAF/Axes/m_h
//     PlcTask Inputs/Main.M8.Axis.NcToPlc <-> Outputs/ToPlc
//     PlcTask Outputs/Main.M8.Axis.PlcToNc <-> Inputs/FromPlc
//   rixs_optics Instance <-> NC-Task 1 SAF/Axes/m_pi
//     PlcTask Inputs/Main.M6.Axis.NcToPlc <-> Outputs/ToPlc
//     PlcTask Outputs/Main.M6.Axis.PlcToNc <-> Inputs/FromPlc
//   rixs_optics Instance <-> NC-Task 1 SAF/Axes/s_io
//     PlcTask Inputs/Main.M10.Axis.NcToPlc <-> Outputs/ToPlc
//     PlcTask Outputs/Main.M10.Axis.PlcToNc <-> Inputs/FromPlc
//   rixs_optics Instance <-> NC-Task 1 SAF/Axes/s_r
//     PlcTask Inputs/Main.M11.Axis.NcToPlc <-> Outputs/ToPlc
//     PlcTask Outputs/Main.M11.Axis.PlcToNc <-> Inputs/FromPlc

// ---- GVLs/Main.TcGVL
VAR_GLOBAL
(*
    Only includes motor definitions for the IOC
    These are hard-coded to be Main.M#,
    but are very convenient to store in a GVL,
    hence the confusing namespace here

    This should be refactored once the IOC
    supports arbitrary ads paths for motors
*)
	(*MR1K2*)
	// Motors
	{attribute 'TcLinkTo' := '.bLimitForwardEnable:=TIIB[EL7047_M1K2_Yleft]^STM Status^Status^Digital input 1;
                              .bLimitBackwardEnable:=TIIB[EL7047_M1K2_Yleft]^STM Status^Status^Digital input 2'}
	{attribute 'pytmc' := '
		pv: MR1K2:SWITCH:MMS:YLEFT
	'}
	M1 : DUT_MotionStage := (fVelocity:=100.0, nEnableMode:=ENUM_StageEnableMode.ALWAYS, bPowerSelf:=True); // M1K2 Yleft
	fbMotionStage_m1 : FB_MotionStage;

	{attribute 'TcLinkTo' := '.bLimitForwardEnable:=TIIB[EL7047_M1K2_Yright]^STM Status^Status^Digital input 1;
                              .bLimitBackwardEnable:=TIIB[EL7047_M1K2_Yright]^STM Status^Status^Digital input 2'}
	{attribute 'pytmc' := '
		pv: MR1K2:SWITCH:MMS:YRIGHT
	'}
	M2 : DUT_MotionStage := (fVelocity:=100.0, nEnableMode:=ENUM_StageEnableMode.ALWAYS, bPowerSelf:=True); // M1K2 Yright
	fbMotionStage_m2 : FB_MotionStage;

	{attribute 'TcLinkTo' := '.bLimitForwardEnable:=TIIB[EL7047_M1K2_Xup]^STM Status^Status^Digital input 1;
                              .bLimitBackwardEnable:=TIIB[EL7047_M1K2_Xup]^STM Status^Status^Digital input 2'}
	{attribute 'pytmc' := '
		pv: MR1K2:SWITCH:MMS:XUP
	'}
	M3 : DUT_MotionStage := (fVelocity:=150.0, nEnableMode:=ENUM_StageEnableMode.ALWAYS, bPowerSelf:=True); // M1K2 Xup
	fbMotionStage_m3 : FB_MotionStage;

	{attribute 'TcLinkTo' := '.bLimitForwardEnable:=TIIB[EL7047_M1K2_Xdwn]^STM Status^Status^Digital input 1;
                              .bLimitBackwardEnable:=TIIB[EL7047_M1K2_Xdwn]^STM Status^Status^Digital input 2'}
	{attribute 'pytmc' := '
		pv: MR1K2:SWITCH:MMS:XDWN
	'}
	M4 : DUT_MotionStage := (fVelocity:=150.0, nEnableMode:=ENUM_StageEnableMode.ALWAYS, bPowerSelf:=True); // M1K2 Xdwn
	fbMotionStage_m4 : FB_MotionStage;

	{attribute 'TcLinkTo' := '.bLimitForwardEnable:=TIIB[EL7047_M1K2_PitchCoarse]^STM Status^Status^Digital input 1;
                              .bLimitBackwardEnable:=TIIB[EL7047_M1K2_PitchCoarse]^STM Status^Status^Digital input 2'}
	{attribute 'pytmc' := '
		pv: MR1K2:SWITCH:MMS:PITCH
	'}
	M5 : DUT_MotionStage := (fVelocity:=30.0, nEnableMode:=ENUM_StageEnableMode.DURING_MOTION, bPowerSelf:=True); // M1K2 Pitch Stepper

	
	(*SP1K1-Mono*)
	{attribute 'pytmc' := '
		pv: SP1K1:MONO:MMS:M_PI
	'}
	{attribute 'TcLinkTo' := '.bLimitForwardEnable:=TIIB[m_pi_m]^STM Status^Status^Digital input 1;
                              .bLimitBackwardEnable:=TIIB[m_pi_m]^STM Status^Status^Digital input 2'}
	M6: DUT_MotionStage:=(nEnableMode:=ENUM_StageEnableMode.DURING_MOTION, fVelocity:=200.0, bPowerSelf:=True); // M_PI, urad
	{attribute 'pytmc' := '
		pv: SP1K1:MONO:MMS:G_PI
	'}
	{attribute 'TcLinkTo' := '.bLimitForwardEnable:=TIIB[g_pi_m]^STM Status^Status^Digital input 1;
                              .bLimitBackwardEnable:=TIIB[g_pi_m]^STM Status^Status^Digital input 2'}
	M7: DUT_MotionStage:=(nEnableMode:=ENUM_StageEnableMode.DURING_MOTION, fVelocity:=200.0, bPowerSelf:=True); // G_PI, urad
	{attribute 'pytmc' := '
		pv: SP1K1:MONO:MMS:M_H
	'}
	{attribute 'TcLinkTo' := '.bLimitForwardEnable:=TIIB[m_h_m]^STM Status^Status^Digital input 1;
                              .bLimitBackwardEnable:=TIIB[m_h_m]^STM Status^Status^Digital input 2'}
	M8: DUT_MotionStage:=(nEnableMode:=ENUM_StageEnableMode.DURING_MOTION, fVelocity:=500.0, bPowerSelf:=True); // M_H, um
	{attribute 'pytmc' := '
		pv: SP1K1:MONO:MMS:G_H
	'}
	{attribute 'TcLinkTo' := '.bLimitForwardEnable:=TIIB[g_h_m]^STM Status^Status^Digital input 1;
                              .bLimitBackwardEnable:=TIIB[g_h_m]^STM Status^Status^Digital input 2'}
	M9: DUT_MotionStage:=(nEnableMode:=ENUM_StageEnableMode.DURING_MOTION, fVelocity:=1000.0, bPowerSelf:=True); // G_H, um
	{attribute 'pytmc' := '
		pv: SP1K1:MONO:MMS:SD_V
	'}
	{attribute 'TcLinkTo' := '.bLimitForwardEnable:=TIIB[s_io_m]^STM Status^Status^Digital input 1;
                              .bLimitBackwardEnable:=TIIB[s_io_m]^STM Status^Status^Digital input 2'}
	M10: DUT_MotionStage:=(nEnableMode:=ENUM_StageEnableMode.DURING_MOTION, fVelocity:=500.0, bPowerSelf:=True); // SD_V, um
	{attribute 'pytmc' := '
		pv: SP1K1:MONO:MMS:SD_ROT
	'}
	// no limits on this motion
	M11: DUT_MotionStage:=(nEnableMode:=ENUM_StageEnableMode.DURING_MOTION, fVelocity:=500.0, bPowerSelf:=True); // SD_R, urad

	(*MR1K1*)
	// Should move before MR1K2 and re-number each motor, lots of work
    // need to fix Axis IDs for IOC to work
	// For now just want functional PLC project
	// Motors
	{attribute 'TcLinkTo' := '.bLimitForwardEnable:=TIIB[EL7047_M1K1_Yup]^STM Status^Status^Digital input 1;
                              .bLimitBackwardEnable:=TIIB[EL7047_M1K1_Ydwn]^STM Status^Status^Digital input 2
								'}
	{attribute 'pytmc' := '
		pv: MR1K1:BEND:MMS:YUP
	'}
	M12 : DUT_MotionStage := (fVelocity:=100.0, nEnableMode:=ENUM_StageEnableMode.ALWAYS, bPowerSelf:=True); // M1K1 Yup
	fbMotionStage_m12 : FB_MotionStage;

	{attribute 'TcLinkTo' := '.bLimitForwardEnable:=TIIB[EL7047_M1K1_Ydwn]^STM Status^Status^Digital input 1;
                              .bLimitBackwardEnable:=TIIB[EL7047_M1K1_Ydwn]^STM Status^Status^Digital input 2'}
	{attribute 'pytmc' := '
		pv: MR1K1:BEND:MMS:YDWN
	'}
	M13 : DUT_MotionStage := (fVelocity:=100.0, nEnableMode:=ENUM_StageEnableMode.ALWAYS, bPowerSelf:=True); // M1K1 Ydwn
	fbMotionStage_m13 : FB_MotionStage;

	{attribute 'TcLinkTo' := '.bLimitForwardEnable:=TIIB[EL7047_M1K1_Xup]^STM Status^Status^Digital input 1;
                              .bLimitBackwardEnable:=TIIB[EL7047_M1K1_Xup]^STM Status^Status^Digital input 2'}
	{attribute 'pytmc' := '
		pv: MR1K1:BEND:MMS:XUP
	'}
	M14 : DUT_MotionStage := (fVelocity:=150.0, nEnableMode:=ENUM_StageEnableMode.ALWAYS, bPowerSelf:=True); // M1K1 Xup
	fbMotionStage_m14 : FB_MotionStage;

	{attribute 'TcLinkTo' := '.bLimitForwardEnable:=TIIB[EL7047_M1K1_Xdwn]^STM Status^Status^Digital input 1;
                              .bLimitBackwardEnable:=TIIB[EL7047_M1K1_Xdwn]^STM Status^Status^Digital input 2'}
	{attribute 'pytmc' := '
		pv: MR1K1:BEND:MMS:XDWN
	'}
	M15 : DUT_MotionStage := (fVelocity:=150.0, nEnableMode:=ENUM_StageEnableMode.ALWAYS, bPowerSelf:=True); // M1K1 Xdwn
	fbMotionStage_m15 : FB_MotionStage;

	{attribute 'TcLinkTo' := '.bLimitForwardEnable:=TIIB[EL7047_M1K1_PitchCoarse]^STM Status^Status^Digital input 1;
                              .bLimitBackwardEnable:=TIIB[EL7047_M1K1_PitchCoarse]^STM Status^Status^Digital input 2'}
	{attribute 'pytmc' := '
		pv: MR1K1:BEND:MMS:PITCH
	'}
	M16 : DUT_MotionStage := (fVelocity:=30.0, nEnableMode:=ENUM_StageEnableMode.DURING_MOTION, bPowerSelf:=True); // M1K1 Pitch Stepper
		
	{attribute 'TcLinkTo' := '.bLimitForwardEnable :=TIIB[EL7041_M1K1_BEND_US]^STM Status^Status^Digital input 1;
                              .bLimitBackwardEnable:=TIIB[EL7041_M1K1_BEND_US]^STM Status^Status^Digital input 2;
							  .nRawEncoderULINT    := TIIB[EL5042_M1K1_BEND_USDS]^FB Inputs Channel 1^Position'}
	{attribute 'pytmc' := '
	pv: MR1K1:BEND:MMS:US
	'}
	M17 : DUT_MotionStage := (nEnableMode:=ENUM_StageEnableMode.DURING_MOTION, bPowerSelf:=TRUE); //MR1K1 US BEND
	fbMotionStage_m17 : FB_MotionStage;
	
	{attribute 'TcLinkTo' := '.bLimitForwardEnable :=TIIB[EL7041_M1K1_BEND_DS]^STM Status^Status^Digital input 1;
                              .bLimitBackwardEnable:=TIIB[EL7041_M1K1_BEND_DS]^STM Status^Status^Digital input 2;
							  .nRawEncoderULINT    := TIIB[EL5042_M1K1_BEND_USDS]^FB Inputs Channel 2^Position'}
	{attribute 'pytmc' := '
	pv: MR1K1:BEND:MMS:DS
	'}
	M18 : DUT_MotionStage := (nEnableMode:=ENUM_StageEnableMode.DURING_MOTION, bPowerSelf:=TRUE); //MR1K1 DS BEND
	fbMotionStage_m18 : FB_MotionStage;
	
	(*SL1K2*)
	// Motors
	{attribute 'TcLinkTo' := '.bLimitForwardEnable:=TIIB[EL7047_SL1K2_PITCH]^STM Status^Status^Digital input 2;
                              .bLimitBackwardEnable:=TIIB[EL7047_SL1K2_PITCH]^STM Status^Status^Digital input 1;
		 					  .nRawEncoderUINT      := TIIB[EL5042_SL1K2_PITCH_VERT]^FB Inputs Channel 1^Position'}
	{attribute 'pytmc' := '
		pv: SL1K2:EXIT:MMS:PITCH
	'}
	M19 : DUT_MotionStage := (sName:= 'SL1K2:EXIT:MMS:PITCH',fVelocity :=0.12);// Air Pitch

	{attribute 'TcLinkTo' := '.bLimitForwardEnable:=TIIB[EL7047_SL1K2_VERT]^STM Status^Status^Digital input 1;
                              .bLimitBackwardEnable:=TIIB[EL7047_SL1K2_VERT]^STM Status^Status^Digital input 2;
		 					  .nRawEncoderUINT      := TIIB[EL5042_SL1K2_PITCH_VERT]^FB Inputs Channel 2^Position'}
	{attribute 'pytmc' := '
		pv: SL1K2:EXIT:MMS:VERT
	'}
	M20 : DUT_MotionStage := (sName:= 'SL1K2:EXIT:MMS:VERT',fVelocity :=0.3); // Air Vertical

	{attribute 'TcLinkTo' := '.bLimitForwardEnable:=TIIB[EL7047_SL1K2_ROLL]^STM Status^Status^Digital input 2;
                              .bLimitBackwardEnable:=TIIB[EL7047_SL1K2_ROLL]^STM Status^Status^Digital input 1;
							  .nRawEncoderUINT      := TIIB[EL5042_SL1K2_ROLL_GAP]^FB Inputs Channel 1^Position'}
	{attribute 'pytmc' := '
		pv: SL1K2:EXIT:MMS:ROLL
	'}
	M21 : DUT_MotionStage := (sName:= 'SL1K2:EXIT:MMS:ROLL',fVelocity :=0.24); // Air Roll

	{attribute 'TcLinkTo' := '.bLimitForwardEnable:=TIIB[EL7047_SL1K2_GAP]^STM Status^Status^Digital input 2;
                              .bLimitBackwardEnable:=TIIB[EL7047_SL1K2_GAP]^STM Status^Status^Digital input 1;
							  .nRawEncoderUINT      := TIIB[EL5042_SL1K2_ROLL_GAP]^FB Inputs Channel 2^Position'}
	{attribute 'pytmc' := '
		pv: SL1K2:EXIT:MMS:GAP
	'}
	M22 : DUT_MotionStage := (sName:= 'SL1K2:EXIT:MMS:GAP',fVelocity :=0.1); // GAP

	{attribute 'TcLinkTo' := '.bLimitForwardEnable:=TIIB[EL7047_SL1K2_YAG]^STM Status^Status^Digital input 1;
                              .bLimitBackwardEnable:=TIIB[EL7047_SL1K2_YAG]^STM Status^Status^Digital input 2;
							  .nRawEncoderUINT      := TIIB[EL5042_SL1K2_YAG]^FB Inputs Channel 1^Position'}
	{attribute 'pytmc' := '
		pv: SL1K2:EXIT:MMS:YAG
	'}
	M23 : DUT_MotionStage := (sName:= 'SL1K2:EXIT:MMS:YAG',fVelocity :=0.5); // YAG
	
	
    // ST1K1-ZOS-MMS
    {attribute 'pytmc' := 'pv: ST1K1:ZOS:MMS'}
    {attribute 'TcLinkTo' := '.bLimitForwardEnable  := TIIB[ST1K1-EL7041]^STM Status^Status^Digital input 1;
                              .bLimitBackwardEnable := TIIB[ST1K1-EL7041]^STM Status^Status^Digital input 2;
                              .bBrakeRelease        := TIIB[ST1K1-EL2008]^Channel 1^Output'}
    M24: DUT_MotionStage := (sName := 'ST1K1:ZOS:MMS');

	
	
	
	sio_current AT%I* : UINT;
	
	sio_load AT%I* : UINT;
	dummyBool: BOOL;
END_VAR

// ---- POUs/PRG_SPO_PMPS.TcPOU
PROGRAM PRG_SPO_PMPS
VAR
	// PMPS
    ffMR1K1Height : FB_FastFault := (
        i_xAutoReset := TRUE,
        i_DevName := 'MR1K1 Height',
        i_Desc := 'MR1K1 Height is out of Single Point Operation safe range',
        i_TypeCode := 16#F501);	
    ffMR1K1Pitch : FB_FastFault := (
        i_xAutoReset := TRUE,
        i_DevName := 'MR1K1 Pitch',
        i_Desc := 'MR1K1 Pitch is out of Single Point Operation safe range',
        i_TypeCode := 16#F502);	
		
    ffSP1K1MPitch : FB_FastFault := (
        i_xAutoReset := TRUE,
        i_DevName := 'SP1K1 Mirror Pitch',
        i_Desc := 'SP1K1 Mirror Pitch is out of Single Point Operation safe range',
        i_TypeCode := 16#F503);	
	ffSP1K1GPitch : FB_FastFault := (
        i_xAutoReset := TRUE,
        i_DevName := 'SP1K1 Grating Pitch',
        i_Desc := 'SP1K1 Grating Pitch is out of Single Point Operation safe range',
        i_TypeCode := 16#F504);	
	ffSP1K1GHorisontal : FB_FastFault := (
        i_xAutoReset := TRUE,
        i_DevName := 'SP1K1 Grating horizontal',
        i_Desc := 'SP1K1 horizontal Pitch is out of Single Point Operation safe range',
        i_TypeCode := 16#F505);		
	
	ffZos : FB_FastFault := (
        i_xAutoReset := TRUE,
        i_DevName := 'T1K1 ZOS',
        i_Desc := 'ST1K1 ZOS is out of Single Point Operation safe range',
        i_TypeCode := 16#F506);	
END_VAR
VAR CONSTANT
	nUpperMR1K1Height : UDINT := 32961458; //POS 32911458+ Delta 50000;
	nLowerMR1K1Height : UDINT := 32861458; //POS 32911458- Delta 50000;
	
	nUpperMR1K1Pitch : UDINT := 10114377;// 10093885 + 20491;
	nLowerMR1K1Pitch : UDINT := 10073393; //10093885 - 20491;
	
	nUpperSP1K1MPitch : UDINT := 31769145;// 31758046 + 11098;
	nLowerSP1K1MPitch : UDINT := 31746947;//31758046 - 11098;
	
	
	nUpperSP1K1GPitch : UDINT := 23624881;
	
	nUpperSP1K1GH: UDINT := 40000000;
	nLowerSP1K1GH: UDINT := 24000000;
	
	nZOSLower : UDINT := 0; // value still needs to be calculated
	
	
END_VAR


//MR1K1 height
ffMR1K1Height.i_xOK := (M12.nEncoderCount > nLowerMR1K1Height ) AND (M12.nEncoderCount < nUpperMR1K1Height );
ffMR1K1Height(io_fbFFHWO := GVL_PMPS.fbFastFaultOutput1);
//MR1K1 pitch
ffMR1K1Pitch.i_xOK := (M16.nEncoderCount > nLowerMR1K1Pitch) AND ( M16.nEncoderCount < nUpperMR1K1Pitch);
ffMR1K1Pitch(io_fbFFHWO := GVL_PMPS.fbFastFaultOutput1);
//SP1K1 mirror pitch
ffSP1K1MPitch.i_xOK := (M6.nEncoderCount > nLowerSP1K1MPitch) AND (M6.nEncoderCount < nUpperSP1K1MPitch); 
ffSP1K1MPitch(io_fbFFHWO := GVL_PMPS.fbFastFaultOutput1);
//SP1K1 grating pitch
ffSP1K1GPitch.i_xOK := (M7.nEncoderCount < nUpperSP1K1GPitch);
ffSP1K1GPitch(io_fbFFHWO := GVL_PMPS.fbFastFaultOutput1);
//SP1K1 Grating horizontal
ffSP1K1GHorisontal.i_xOK := (M9.nEncoderCount > nLowerSP1K1GH) AND (M9.nEncoderCount < nUpperSP1K1GH); 
ffSP1K1GHorisontal(io_fbFFHWO := GVL_PMPS.fbFastFaultOutput1);
//ST1K1 ZOS
ffZos.i_xOK := M24.nEncoderCount > nZOSLower;
ffZos(io_fbFFHWO := GVL_PMPS.fbFastFaultOutput1);

END_PROGRAM
